(* PLC project Sem nome, Desconhecido Sem nome 1 *)
(* stored: creationDateTime 2022-02-11T07:24:12, modificationDateTime 2022-02-12T11:21:20 *)

PROGRAM Controle_Servo
  VAR
    START AT %IX100.0 : BOOL;
    STOP AT %IX100.1 : BOOL;
    CONTROL AT %IX100.2 : BOOL;
    START_LED AT %QX100.0 : BOOL;
    STOP_LED AT %QX100.1 : BOOL := True;
    OUTPUT AT %QX100.2 : BOOL;
  END_VAR
  VAR
    TON0 : TON;
  END_VAR
  VAR
    ENABLE_CONTROL AT %MX100 : BOOL;
  END_VAR

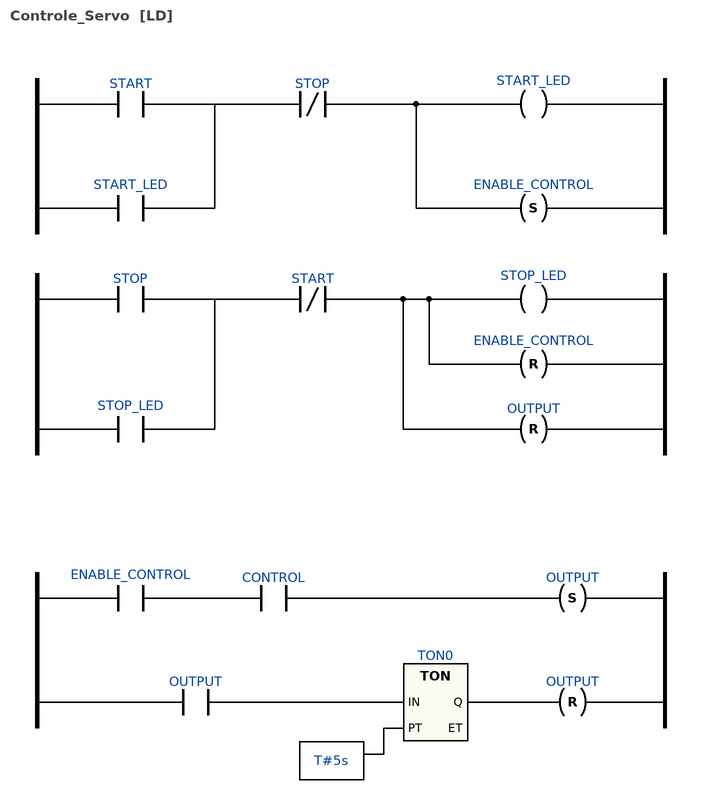
(* LD diagram, written out as Structured Text *)
START_LED := (START OR START_LED) AND NOT STOP;
IF (START OR START_LED) AND NOT STOP THEN ENABLE_CONTROL := TRUE; END_IF;
STOP_LED := (STOP OR STOP_LED) AND NOT START;
IF (STOP OR STOP_LED) AND NOT START THEN ENABLE_CONTROL := FALSE; END_IF;
IF (STOP OR STOP_LED) AND NOT START THEN OUTPUT := FALSE; END_IF;
IF ENABLE_CONTROL AND CONTROL THEN OUTPUT := TRUE; END_IF;
TON0(IN := OUTPUT, PT := T#5s);
IF TON0.Q THEN OUTPUT := FALSE; END_IF;
END_PROGRAM

CONFIGURATION Config0
  RESOURCE Res0 ON PLC
    TASK task0(INTERVAL := T#20ms, PRIORITY := 0);
    PROGRAM instance0 WITH task0 : Controle_Servo;
  END_RESOURCE
END_CONFIGURATION
